FUNCTION_BLOCK OutputLogger (* Extracted Composite Function Block Type *)
  (* Version 11/3/2016, chivdan *)
  PACKAGE Main;
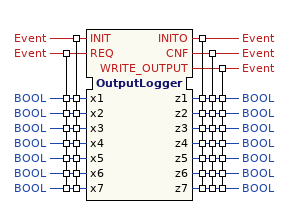
  EVENT_INPUT
    INIT WITH x1, x2, x3, x4, x5, x6, x7; (* Initialization request *)
    REQ WITH x1, x2, x3, x4, x5, x6, x7; (* Normal Execution Request *)
  END_EVENT
  EVENT_OUTPUT
    INITO WITH z1, z2, z3, z4, z5, z6, z7; (* Initialization confirmation event *)
    CNF WITH z1, z2, z3, z4, z5, z6, z7; (* Log request confirmation *)
    WRITE_OUTPUT WITH z1, z2, z3, z4, z5, z6, z7; (* Execution Confirmation *)
  END_EVENT
  VAR_INPUT
    x1 : BOOL; (* Argument *)
    x2 : BOOL; (* Argument *)
    x3 : BOOL; (* Argument *)
    x4 : BOOL; (* Argument *)
    x5 : BOOL; (* Argument *)
    x6 : BOOL; (* Argument *)
    x7 : BOOL; (* Argument *)
  END_VAR
  VAR_OUTPUT
    z1 : BOOL;
    z2 : BOOL;
    z3 : BOOL;
    z4 : BOOL;
    z5 : BOOL;
    z6 : BOOL;
    z7 : BOOL;
  END_VAR
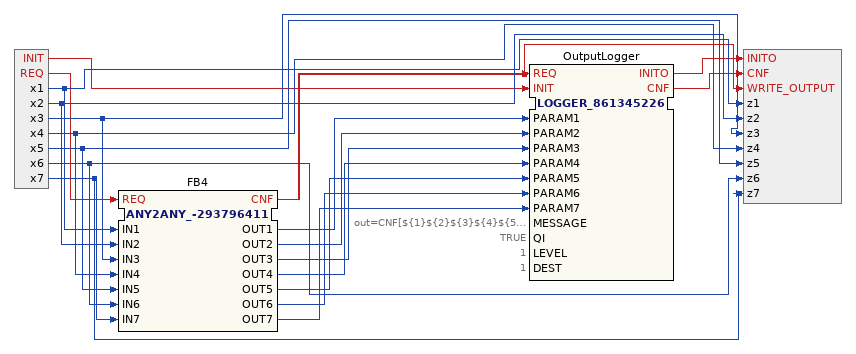
  FBS
    OutputLogger : LOGGER_861345226(MESSAGE := out=CNF[${1}${2}${3}${4}${5}${6}${7}], QI := TRUE, LEVEL := 1, DEST := 1); {SET_ATTRIBUTE(Configuration.GenericFBType.InterfaceParams, Runtime.System#CNT:=7)}
    FB4 : ANY2ANY_-293796411; {SET_ATTRIBUTE(Configuration.GenericFBType.InterfaceParams, Runtime.Standard#CNT:=7;IN${CNT$}:BOOL,BOOL,BOOL,BOOL,BOOL,BOOL,BOOL;OUT${CNT$}:INT,INT,INT,INT,INT,INT,INT)}
  END_FBS
  EVENT_CONNECTIONS
    FB4.CNF TO OutputLogger.REQ;
    REQ TO FB4.REQ;
    OutputLogger.INITO TO INITO;
    OutputLogger.CNF TO CNF;
    INIT TO OutputLogger.INIT;
    FB4.CNF TO WRITE_OUTPUT;
  END_CONNECTIONS
  DATA_CONNECTIONS
    FB4.OUT1 TO OutputLogger.PARAM1;
    FB4.OUT2 TO OutputLogger.PARAM2;
    FB4.OUT3 TO OutputLogger.PARAM3;
    FB4.OUT4 TO OutputLogger.PARAM4;
    FB4.OUT5 TO OutputLogger.PARAM5;
    FB4.OUT6 TO OutputLogger.PARAM6;
    FB4.OUT7 TO OutputLogger.PARAM7;
    x1 TO FB4.IN1;
    x2 TO FB4.IN2;
    x3 TO FB4.IN3;
    x4 TO FB4.IN4;
    x5 TO FB4.IN5;
    x6 TO FB4.IN6;
    x7 TO FB4.IN7;
    x1 TO z1;
    x2 TO z2;
    x3 TO z3;
    x4 TO z4;
    x5 TO z5;
    x6 TO z6;
    x7 TO z7;
  END_CONNECTIONS
END_FUNCTION_BLOCK
